{attribute 'linkalways'} 
{attribute 'no_explicit_call' := 'This FB is a CLASS and must be accessed using methods or properties'}
{attribute 'enable_dynamic_creation'}
FUNCTION_BLOCK _ETcVnDrawShape EXTENDS EnumDatatypeBase
VAR
	localData : ETcVnDrawShape;
	activeData : REFERENCE TO ETcVnDrawShape;
	enumBaseDatatype : _DINT(localData);
END_VAR

METHOD PRIVATE AddLocalEnumeration
VAR_INPUT
	Enumeration : T_MAXSTRING;
	Value : ETcVnDrawShape;
END_VAR
AddEnumeration(Enumeration, Value);
END_METHOD

PROPERTY PUBLIC Address : PVOID
GET
Address := ADR(activeData);
END_GET
END_PROPERTY

METHOD PUBLIC ClearReference
VAR_INPUT
END_VAR
activeData REF= localData;
SetBaseDatatypeReference();
END_METHOD

METHOD PUBLIC Clone : I_Datatype
VAR
    pClone : POINTER TO _ETcVnDrawShape;
END_VAR
pClone := __NEW(_ETcVnDrawShape(InitialValue := Value));
Clone := pClone^;
END_METHOD

METHOD FB_init : BOOL
VAR_INPUT
	bInitRetains : BOOL; // if TRUE, the retain variables are initialized (warm start / cold start)
	bInCopyCode : BOOL;  // if TRUE, the instance afterwards gets moved into the copy code (online change)
	InitialValue : ETcVnDrawShape;
END_VAR
localData := InitialValue;
AddBaseDatatype(enumBaseDatatype);
ClearReference();

AddLocalEnumeration('TCVN_DS_RANDOM', ETcVnDrawShape.TCVN_DS_RANDOM);
AddLocalEnumeration('TCVN_DS_CIRCLE', ETcVnDrawShape.TCVN_DS_CIRCLE);
AddLocalEnumeration('TCVN_DS_SQUARE', ETcVnDrawShape.TCVN_DS_SQUARE);
AddLocalEnumeration('TCVN_DS_PLUS', ETcVnDrawShape.TCVN_DS_PLUS);
AddLocalEnumeration('TCVN_DS_X', ETcVnDrawShape.TCVN_DS_X);
AddLocalEnumeration('TCVN_DS_DIAMOND', ETcVnDrawShape.TCVN_DS_DIAMOND);
AddLocalEnumeration('TCVN_DS_MAX', ETcVnDrawShape.TCVN_DS_MAX);
END_METHOD

PROPERTY PUBLIC Identifier : T_MAXSTRING
GET
Identifier := 'ETcVnDrawShape';
END_GET
END_PROPERTY

METHOD IsEnumeratorValueEqual : BOOL
VAR_INPUT
	Enumerator : I_KeyValueForwardEnumerator;
END_VAR
VAR
	storedValue : ETcVnDrawShape;
END_VAR
IF NOT Enumerator.TryGet(storedValue) THEN
	RETURN;
END_IF

IsEnumeratorValueEqual := storedValue = activeData;
END_METHOD

METHOD PUBLIC MakeReferenceTo
VAR_INPUT
	ReferenceTarget : REFERENCE TO ETcVnDrawShape;
END_VAR
activeData REF= ReferenceTarget;
SetBaseDatatypeReference();
END_METHOD

METHOD PROTECTED SetBaseDatatypeReference
VAR_INPUT
END_VAR
enumBaseDatatype.MakeReferenceTo(activeData);
END_METHOD

PROPERTY PUBLIC Size : UDINT
GET
Size := SIZEOF(activeData);
END_GET
END_PROPERTY

METHOD TryMakeReferenceTo : BOOL
VAR_INPUT
	Target : I_Datatype;
END_VAR
VAR
	targetAsEnum : I_EnumDatatype;
	pTargetData : POINTER TO ETcVnDrawShape;
END_VAR
IF NOT Target.TryResolveAsEnumDatatype(targetAsEnum) THEN
	RETURN;
END_IF

IF targetAsEnum.Identifier <> Identifier THEN
	RETURN;
END_IF

pTargetData := Target.Address;
activeData REF= pTargetData^;
SetBaseDatatypeReference();
TryMakeReferenceTo := TRUE;
END_METHOD

PROPERTY PUBLIC Value : ETcVnDrawShape
GET
Value := activeData;
END_GET
SET
activeData := Value;
END_SET
END_PROPERTY

END_FUNCTION_BLOCK

(* stored: Version 1.1.0.1, ProductVersion 3.1.4024.12
   POU _ETcVnDrawShape: Id {b8fa2840-ad1b-4681-a66c-9cd387b557d4}, SpecialFunc None
   Folder Constructor: Id {edfe3b8c-39f9-48fb-96e6-79af75f555af}
   Folder Private: Id {c655dfcb-e87b-47a1-97c2-2e6aa35af10a}
   Folder Protected: Id {a5ebba3b-f2c1-48ce-9958-19d5f5c6a406}
   Method AddLocalEnumeration: Id {6e714d31-63f7-42fa-825b-cda8edffb4d7}
   Property Address: Id {fa3a0a41-50d4-4ea9-a5e5-0bf63bfdd0c3}
   Get Get: Id {f33a2b7a-107f-4888-99c8-2f9db9707145}
   Method ClearReference: Id {5f5e1bd8-6c47-47a5-8358-3cdb86f3740b}
   Method Clone: Id {34f53c88-50da-46bb-be00-dbf767f333a7}
   Method FB_init: Id {0a0ef9d2-9c2b-462b-8a56-82223c02f7fb}
   Property Identifier: Id {5bbc03c7-c7a9-4dba-bca8-1ccb3686ff6b}
   Get Get: Id {79591d9b-4d90-4923-bb5d-039db1c0f578}
   Method IsEnumeratorValueEqual: Id {88cd2a7d-a273-4b94-9d30-dd428d609e52}
   Method MakeReferenceTo: Id {2b6a5769-7ccc-4f7b-bb20-aba6ddaffaf8}
   Method SetBaseDatatypeReference: Id {b4996e03-97f6-4494-9d1b-b97479db43ee}
   Property Size: Id {90000892-da81-430d-b39d-39628e4e213a}
   Get Get: Id {d5041247-6938-4080-b479-6013cc64fc32}
   Method TryMakeReferenceTo: Id {e7a56bae-99e5-41ea-adb8-8c3c05abf459}
   Property Value: Id {2928fb2a-7fdd-482a-9dc4-68c500217c69}
   Get Get: Id {d659626e-cac4-45bc-a984-3ba822006ecd}
   Set Set: Id {d94317c9-5603-4fe7-b0ac-f95f3591d0bf} *)
